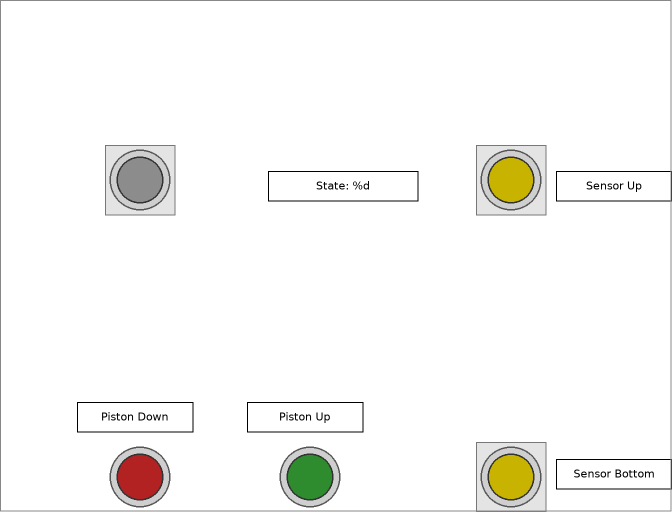
VISUALIZATION Visualization  // 672x512
    PushSwitch (105,145 70x70), variable: MAIN.bStartButton, behaviour: TOGGLE, style: Switch-PushSwitch-Gray
    Lamp1 (105,442 70x70), variable: MAIN.bPistonDown, style: Lamp-Lamp1-Red
    Lamp1 (275,442 70x70), variable: MAIN.bPistonUp, style: Lamp-Lamp1-Green
    Rectangle (268,171 150x30), "State: %d", text variable: MAIN.iState
    Rectangle (77,402 116x30), "Piston Down", text variable: MAIN.iState
    Rectangle (247,402 116x30), "Piston Up", text variable: MAIN.iState
    Rectangle (556,459 116x30), "Sensor Bottom", text variable: MAIN.iState
    Rectangle (556,171 116x30), "Sensor Up", text variable: MAIN.iState
    PushSwitch (476,442 70x70), variable: MAIN.bSensorBottom, behaviour: TOGGLE, style: Switch-PushSwitch-Yellow
    PushSwitch (476,145 70x70), variable: MAIN.bSensorTop, behaviour: TOGGLE, style: Switch-PushSwitch-Yellow
END_VISUALIZATION

(* stored: Version 1.1.0.1
   Visu Visualization: Id {43e63611-ea8c-4cfa-97f7-a44ecd52e68b} *)
